(* PLC project  *)

PROGRAM P
  VAR  (* added by the conversion: wires and edge detectors of the diagram *)
    _ADD3_ENO : BOOL;
    _ADD3_OUT : INT;
    R_TRIG1 : R_TRIG;
  END_VAR

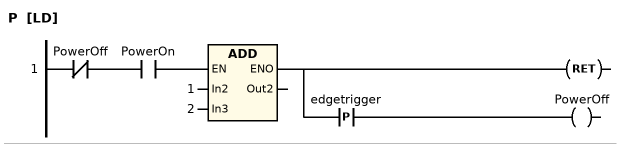
(* LD diagram, written out as Structured Text *)
_ADD3_OUT := ADD(EN := NOT PowerOff AND PowerOn, IN1 := 1, IN2 := 2, ENO => _ADD3_ENO);
IF _ADD3_ENO THEN RETURN; END_IF;
R_TRIG1(CLK := edgetrigger);
PowerOff := _ADD3_ENO AND R_TRIG1.Q;
END_PROGRAM
